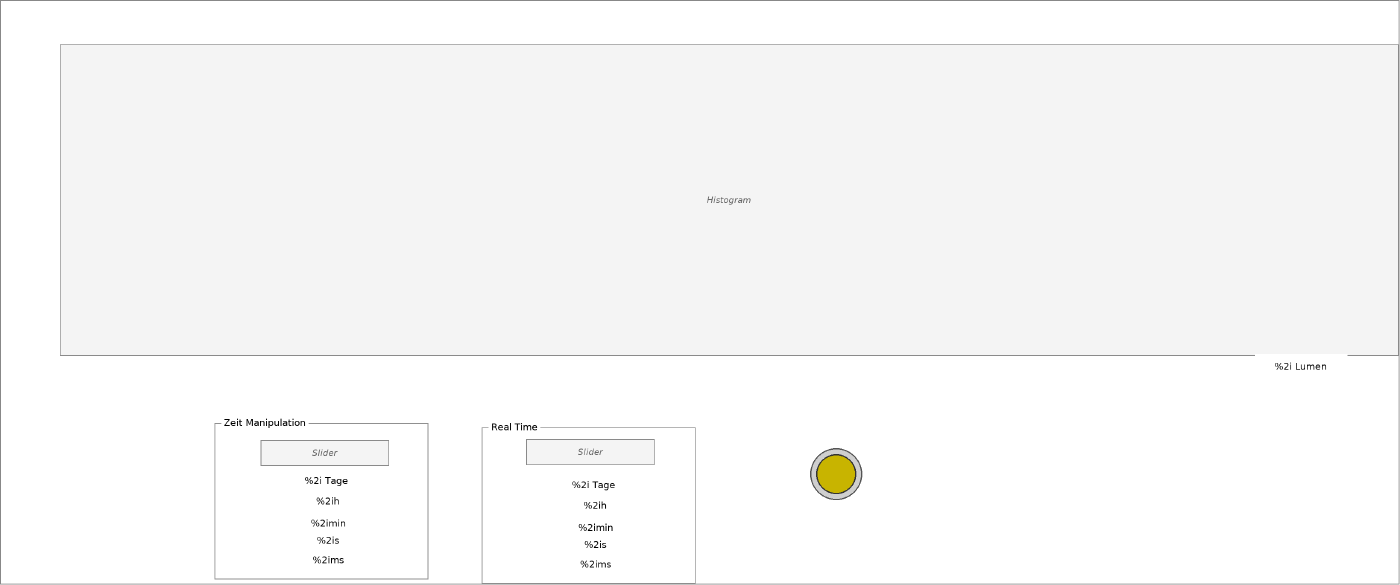
VISUALIZATION Visualization  // 1639x686
    Histogram (70,52 1567x365), scale format: %i, scale 0..3000
        p1518820177: testData
        p102497268: testData
        p788070771: ARRAY [0..50] OF INT
    GroupBox (251,488 250x191), "Zeit Manipulation"
        Slider (54,28 150x30), variable: Zeit_Multiplikator, scale 0..3
        Textfield (102,61 62x30), "%2i Tage", text variable: day
        Textfield (101,111 65x30), "%2imin", text variable: _minute
        Textfield (100,131 66x30), "%2is", text variable: _sekunde
        Textfield (100,154 67x30), "%2ims", text variable: _mSekunde
        Textfield (102,85 62x30), "%2ih", text variable: _stunde
    GroupBox (564,493 250x191), "Real Time"
        Textfield (102,61 62x30), "%2i Tage", text variable: _Rday
        Slider (52,22 150x30), variable: Sin_manipulator, scale 0..3
        Textfield (101,111 65x30), "%2imin", text variable: _Rminute
        Textfield (100,131 66x30), "%2is", text variable: _Rsekunde
        Textfield (100,154 67x30), "%2ims", text variable: _RmSekunde
        Textfield (102,85 62x30), "%2ih", text variable: _Rstunde
    Textfield (1469,415 108x30), "%2i Lumen", text variable: Licht
    Lamp1 (944,521 70x70), variable: Regen, style: Lamp-Lamp1-Yellow
END_VISUALIZATION

(* stored: Version 1.1.0.1, ProductVersion 3.1.4018.5
   Visu Visualization: Id {0236438a-636b-48a4-bb82-1f0497612fc4} *)
